FUNCTION_BLOCK FB_RaiseAlarm
VAR_INPUT
	raiseAlarm: BOOL;
END_VAR
VAR_OUTPUT
END_VAR
VAR
	fbAlarm1: FB_TcAlarm;
	hr1 : HRESULT;
	hr2 : HRESULT;
END_VAR

IF raiseAlarm THEN
	fbAlarm1.CreateEx(TC_Events.MyEventClass.MySecondAlarm, TRUE, 0);
	fbAlarm1.Raise(0);
END_IF

IF fbAlarm1.eConfirmationState = 3 THEN // Waiting for confirmation
	hr1 := fbAlarm1.Clear(0, FALSE); // Veranderd de state niet van Confirmed naar cleared. de state blijft Confirmed
	hr2 := fbAlarm1.Release();  // Zet de state naar NotSupported (0)
END_IF

END_FUNCTION_BLOCK

(* stored: Version 1.1.0.1, ProductVersion 3.1.4022.16
   POU FB_RaiseAlarm: Id {a86e7208-70e1-4801-9566-47af1d00dce2}, SpecialFunc None *)
